(* CoDeSys 2.3 export: FK15PUMPAUTOCONTROL.EXP *)

(* POU K15/fK15PumpAutoControl, ST *)
FUNCTION fK15PumpAutoControl :BOOL
VAR_INPUT
	PumpID : USINT;
	EmergencyPumpStopButtonPressed : BOOL;
END_VAR
VAR
	i: USINT;
END_VAR
(*выключаем все насосы кроме данного*)
FOR i := 1 TO MAX_K15_PUMPS_NUM DO
	IF i <> PumpID THEN
		fTurnOffK15Pump(i);
	END_IF;
END_FOR;

IF EmergencyPumpStopButtonPressed THEN	(*Нажат аварийный стоп насоса?*)
	fTurnOffK15Pump(PumpID); (*Выключить насос*)
	RETURN;
END_IF;

IF K15PumpFaulty[PumpID] THEN
	fTurnOffK15Pump(PumpID); (*Выключить насос*)
ELSE
	fTurnOnK15Pump(PumpID); (*Включить насос*)
END_IF;
END_FUNCTION
